// TIA Portal V20 export
DATA_BLOCK "CallEquipment_DB"   // DB98
{ DB_Accessible_From_OPC_UA := 'FALSE' }
// stored: AssignedProDiagFB Unit1.Em10.ProDiag, DBAccessibleFromOPCUA false, DBAccessibleFromWebserver false, InstanceOfName Unit1.Em10.CallEquipment, InstanceOfType FB, Namespace Unit1.Em10
"Unit1.Em10.CallEquipment"
   // VAR_INPUT
   //    ZoneOperationEnable { ExternalWritable := 'False'} : "LWONIK_typeSafetyZoneManualOperation";
   // END_VAR
   // VAR_IN_OUT
   //    unitStatus : "LAF_typeUnitStatus";
   //    emFeedback : "LUC_typeEmFeedback";
   //    unitAlarmDB : "LAF_typeAlarms";
   // END_VAR
   // VAR
   //    InstSequenceLaserMark { ExternalWritable := 'False'} : "Unit1.Em10.Sequence_1_LaserMark";
   //    instLaserMarkHomeJob1 { ExternalWritable := 'False'} : "LAF_SelectJob";
   //    instLaserMarkLoadJob2 { ExternalWritable := 'False'} : "LAF_SelectJob";
   //    instLaserMarkInspectionJob3 { ExternalWritable := 'False'} : "LAF_SelectJob";
   //    instLaserMarkUnloadJob4 { ExternalWritable := 'False'} : "LAF_SelectJob";
   //    instCmLaserMarkJRDetect { ExternalWritable := 'False'} : "LBC_DigitalSignalCn";
   //    instCmLaserMarkCoverUpDown { ExternalWritable := 'False'} : "LBC_TwoWayActuatorCn";
   //    instCmLaserMarkStageLiftUpDown { ExternalWritable := 'False'} : "LBC_TwoWayActuatorCn";
   //    instLaserMarkControl { ExternalWritable := 'False'} : "LER_LaserMark";
   //    instQrFixReader { ExternalWritable := 'False'} : "LER_QRread_SRX300";
   //    instLaserMarkHistory { ExternalWritable := 'False'} : "LER_laserMarkHistory";
   //    instTraceCodeGeneration { ExternalWritable := 'False'} : "za_TracecodeGeneration";
   //    instManageAlarms { ExternalWritable := 'False'} : "LAF_ManageAlarms";
   //    instEventsPFE { ExternalWritable := 'False'} : "Unit1.Em10.EventsPFE";
   //    statUnitStatus { ExternalWritable := 'False'} : "LAF_typeUnitStatus";
   //    statPartData { ExternalWritable := 'False'} : "LER_typePartData";
   //    statPartData_NG { ExternalWritable := 'False'} : "LER_typePartData";
   //    EmPartData { ExternalWritable := 'False'} : "LER_typePartData";
   //    statDataDelete { ExternalWritable := 'False'} : "LER_typePartData";
   //    statHistoryDeleteData { ExternalWritable := 'False'} : "LER_typeLaserMarkHistory";
   //    statTonTime { ExternalWritable := 'False'} : Array[0..999] of TON_TIME;
   //    statTofTime { ExternalWritable := 'False'} : Array[0..9] of TOF_TIME;
   //    statPulse { ExternalWritable := 'False'} : Array[0..999] of Bool;
   //    statTraceCode { ExternalWritable := 'False'} : Struct
   //       SaveHold : Bool;
   //       ModeOff : Bool;
   //       GenerationBusy_1 : Bool;
   //       GenerationBusy_2 : Bool;
   //       Generation_First : Bool;
   //       Generation_Run_Total : Bool;
   //       SnIncrement_Total : Bool;
   //       SnReset : Bool;
   //       BufferReset : Bool;
   //       "ResultData_Raw[1]" : String[18];
   //       "ResultData_Raw[2]" : String[26];
   //       "ResultData_Raw[3]" : String[5];
   //       ResultData_TC : String[32];
   //       DataSave_1 : Bool;
   //       DataSave_2 : Bool;
   //       Generation_Run_1 : Bool;
   //       SnIncrement_1 : Bool;
   //       Generation_Run_2 : Bool;
   //       SnIncrement_2 : Bool;
   //    END_STRUCT;
   //    statEnableManualCmds { ExternalWritable := 'False'} : Bool;
   //    statNomalMode { ExternalWritable := 'False'} : Bool;
   //    "*** Interlock TwoWay ***" { S7_SetPoint := 'True'} : "LER_Axis_Homing";
   //    instCmLaserMarkCoverUpDownInterlock { S7_SetPoint := 'True'} : Array[0..2] of "LER_Actuator";
   //    instCmLaserMarkStageLiftUpDownInterlock { S7_SetPoint := 'True'} : Array[0..2] of "LER_Actuator";
   //    LaserMarkCoverUpDown_Inpos : Array[0..2] of Struct
   //       "Int" : Array[1..10] of Bool;
   //    END_STRUCT;
   //    LaserMarkStageLiftUpDown_Inpos : Array[0..2] of Struct
   //       "Int" : Array[1..10] of Bool;
   //    END_STRUCT;
   //    citi_Ptrig : Array[0..20] of Bool;
   //    citiTon : Array[0..20] of TON_TIME;
   //    citi : Time;
   //    citiTest : Array[0..20] of Bool;
   // END_VAR
BEGIN
END_DATA_BLOCK
